FUNCTION_BLOCK QUERY_STATION1
  {SET_ATTRIBUTE(OpcUa, SERVICE)}
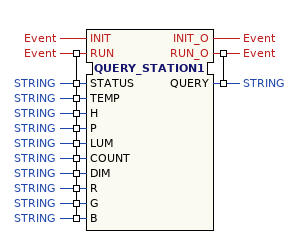
  EVENT_INPUT
    INIT;
    RUN WITH STATUS, TEMP, H, P, LUM, COUNT, DIM, R, G, B; {SET_ATTRIBUTE(OpcUa, Method)}
  END_EVENT
  EVENT_OUTPUT
    INIT_O;
    RUN_O WITH QUERY;
  END_EVENT
  VAR_INPUT
    STATUS : STRING;
    TEMP : STRING;
    H : STRING;
    P : STRING;
    LUM : STRING;
    COUNT : STRING;
    DIM : STRING;
    R : STRING;
    G : STRING;
    B : STRING;
  END_VAR
  VAR_OUTPUT
    QUERY : STRING;
  END_VAR
END_FUNCTION_BLOCK
